{attribute 'Tc2GvlVarNames'}
{attribute 'strict'}
//Riferimento origine assi postazione in WA rispetto l'origine degli assi
TYPE e_RiferimentoPostazione :
(
	NOT_DEFINED			:= -1,
	ANGOLO_DX	 	:= 1,	(* Identifica che IL RISCONTRO della WorkArea è disposta nell'angolo a DX della WorkArea stessa *)
	CENTRALE	 	:= 2,	(* Identifica che IL RISCONTRO della WorkArea è disposta sulla mediana della WorkArea stessa *)	
	ANGOLO_SX	 	:= 3,	(* Identifica che IL RISCONTRO della WorkArea è disposta nell'angolo a SX della WorkArea stessa *)
	XSX_YCENTRALE 	:= 4, 	(* Identifica che IL RISCONTRO della WorkArea è disposta SX della WorkArea stessa MA LASSE Y è IN CENTRO*)
	XDX_YCENTRALE 	:= 5  	(* Identifica che IL RISCONTRO della WorkArea è disposta DX della WorkArea stessa MA LASSE Y è IN CENTRO *)
);
END_TYPE
//  NOT_DEFINED = '-1'

(* stored: Version 1.1.0.1, ProductVersion 3.1.4024.11
   EnumerationTextList e_RiferimentoPostazione: Id {d4f61f88-e658-4899-a3f2-1bb6dc6370a4} *)
